// TIA Portal V21 export
DATA_BLOCK "DateTime"   // DB118
{ S7_Optimized_Access := 'FALSE' }
// stored: AutoNumber false
   VAR
      time_local_read : DTL;
      time_system_read : DTL;
      time_system_write : DTL;
      local_time : Int := 0;
      read_system_time : Int;
      write_system_time : Int;
      write_time : Bool := false;
      write_time_re : Bool;
      time_local_read_ReportName : DTL;
   END_VAR
BEGIN
END_DATA_BLOCK
